// TIA Portal V17 export
// export: Created 2025-03-07T09:17:33.1153197Z, ExportSetting WithDefaults, DisplayName Totally Integrated Automation Portal, DisplayVersion V17 Update 8, DisplayName TIA Portal Openness, DisplayVersion V17 Update 8, DisplayName TIA Portal Version Control Interface, DisplayVersion V17, DisplayName SINAMICS Startdrive Advanced, DisplayVersion V17 SP2, DisplayName SINAMICS Startdrive G110M, G120, G120C, G120D, G120P, G115D, DisplayVersion V17 SP2, DisplayName SINAMICS Startdrive G130, G150, S120, S150, SINAMICS MV, S210, DisplayVersion V17 SP2, DisplayName STEP 7 Professional, DisplayVersion V17 Update 8, DisplayName SINUMERIK ONE STEP 7 Toolbox, DisplayVersion V17 Update 12, DisplayName SINUMERIK 840D sl STEP 7 Toolbox, DisplayVersion V17 Update 12, DisplayName STEP 7 Safety, DisplayVersion V17 Update 6, DisplayName WinCC Advanced, DisplayVersion V17 Update 8
FUNCTION "FC329_CHANNEL_9" : Void   // FC329, LAD
{ S7_Optimized_Access := 'FALSE' }
AUTHOR : ETXETAR
VERSION : 1.0
// stored: AutoNumber false, IsIECCheckEnabled false, SetENOAutomatically false, UDAEnableTagReadback false
   VAR_TEMP
      NC_RESET_CH4 : Bool;
      NC_START_CH4 : Bool;
   END_VAR
BEGIN

REGION Network 1: RESET CHANNEL
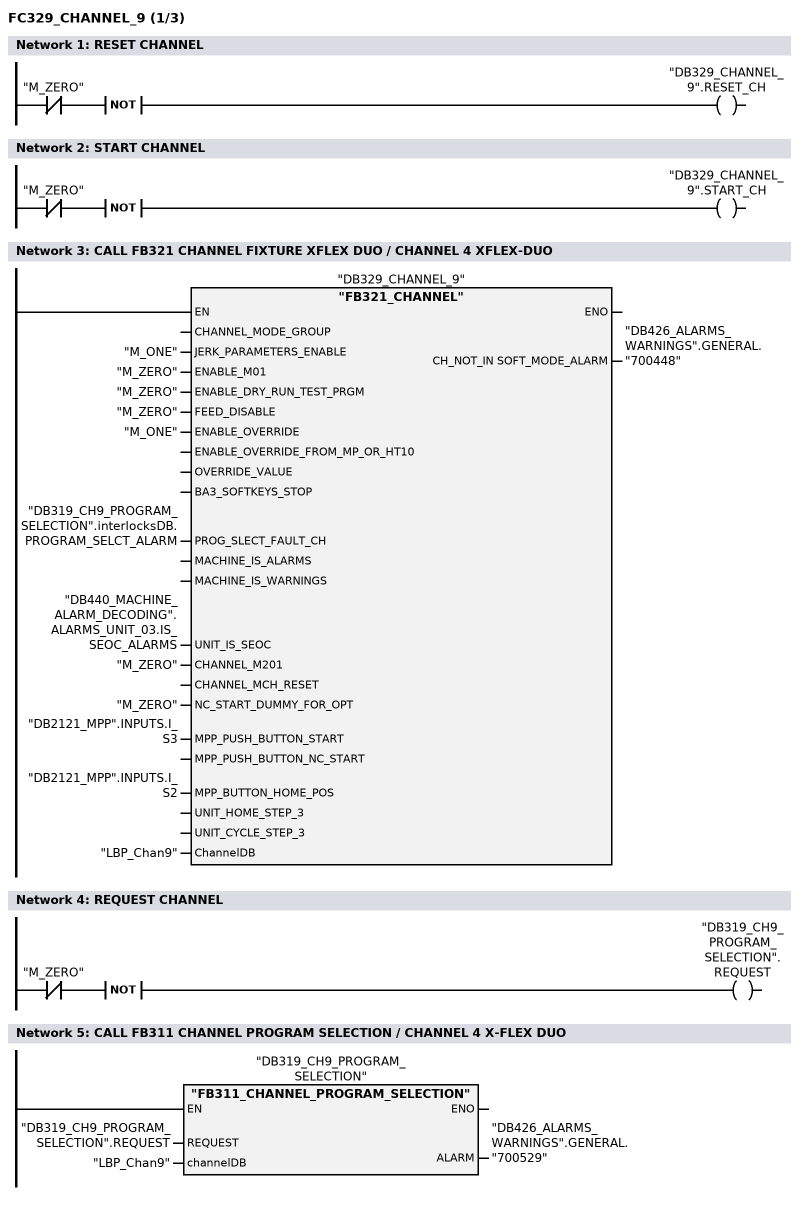
   RUNG wire#powerrail
      I_Contact( "M_ZERO" )
      Not()
      Coil( "DB329_CHANNEL_9".RESET_CH )
   END_RUNG
   // the same network as SCL:
   "DB329_CHANNEL_9".RESET_CH := NOT (NOT "M_ZERO");
END_REGION

REGION Network 2: START CHANNEL
   RUNG wire#powerrail
      I_Contact( "M_ZERO" )
      Not()
      Coil( "DB329_CHANNEL_9".START_CH )
   END_RUNG
   // the same network as SCL:
   "DB329_CHANNEL_9".START_CH := NOT (NOT "M_ZERO");
END_REGION

REGION Network 3: CALL FB321 CHANNEL FIXTURE XFLEX DUO / CHANNEL 4 XFLEX-DUO
   RUNG wire#powerrail
      "DB329_CHANNEL_9"(CHANNEL_MODE_GROUP :=, JERK_PARAMETERS_ENABLE := "M_ONE", ENABLE_M01 := "M_ZERO", ENABLE_DRY_RUN_TEST_PRGM := "M_ZERO", FEED_DISABLE := "M_ZERO", ENABLE_OVERRIDE := "M_ONE", ENABLE_OVERRIDE_FROM_MP_OR_HT10 :=, OVERRIDE_VALUE :=, BA3_SOFTKEYS_STOP :=, PROG_SLECT_FAULT_CH := "DB319_CH9_PROGRAM_SELECTION".interlocksDB.PROGRAM_SELCT_ALARM, MACHINE_IS_ALARMS :=, MACHINE_IS_WARNINGS :=, UNIT_IS_SEOC := "DB440_MACHINE_ALARM_DECODING".ALARMS_UNIT_03.IS_SEOC_ALARMS, CHANNEL_M201 := "M_ZERO", CHANNEL_MCH_RESET :=, NC_START_DUMMY_FOR_OPT := "M_ZERO", MPP_PUSH_BUTTON_START := "DB2121_MPP".INPUTS.I_S3, MPP_PUSH_BUTTON_NC_START :=, MPP_BUTTON_HOME_POS := "DB2121_MPP".INPUTS.I_S2, UNIT_HOME_STEP_3 :=, UNIT_CYCLE_STEP_3 :=, ChannelDB := "LBP_Chan9", "CH_NOT_IN SOFT_MODE_ALARM" => "DB426_ALARMS_WARNINGS".GENERAL."700448")
   END_RUNG
   // the same network as SCL:
   "DB329_CHANNEL_9"(JERK_PARAMETERS_ENABLE := "M_ONE",   // "FB321_CHANNEL"
                     ENABLE_M01 := "M_ZERO",
                     ENABLE_DRY_RUN_TEST_PRGM := "M_ZERO",
                     FEED_DISABLE := "M_ZERO",
                     ENABLE_OVERRIDE := "M_ONE",
                     PROG_SLECT_FAULT_CH := "DB319_CH9_PROGRAM_SELECTION".interlocksDB.PROGRAM_SELCT_ALARM,
                     UNIT_IS_SEOC := "DB440_MACHINE_ALARM_DECODING".ALARMS_UNIT_03.IS_SEOC_ALARMS,
                     CHANNEL_M201 := "M_ZERO",
                     NC_START_DUMMY_FOR_OPT := "M_ZERO",
                     MPP_PUSH_BUTTON_START := "DB2121_MPP".INPUTS.I_S3,
                     MPP_BUTTON_HOME_POS := "DB2121_MPP".INPUTS.I_S2,
                     ChannelDB := "LBP_Chan9",
                     "CH_NOT_IN SOFT_MODE_ALARM" => "DB426_ALARMS_WARNINGS".GENERAL."700448");
END_REGION

REGION Network 4: REQUEST CHANNEL
   RUNG wire#powerrail
      I_Contact( "M_ZERO" )
      Not()
      Coil( "DB319_CH9_PROGRAM_SELECTION".REQUEST )
   END_RUNG
   // the same network as SCL:
   "DB319_CH9_PROGRAM_SELECTION".REQUEST := NOT (NOT "M_ZERO");
END_REGION

REGION Network 5: CALL FB311 CHANNEL PROGRAM SELECTION / CHANNEL 4 X-FLEX DUO
   RUNG wire#powerrail
      "DB319_CH9_PROGRAM_SELECTION"(REQUEST := "DB319_CH9_PROGRAM_SELECTION".REQUEST, channelDB := "LBP_Chan9", ALARM => "DB426_ALARMS_WARNINGS".GENERAL."700529")
   END_RUNG
   // the same network as SCL:
   "DB319_CH9_PROGRAM_SELECTION"(REQUEST := "DB319_CH9_PROGRAM_SELECTION".REQUEST,   // "FB311_CHANNEL_PROGRAM_SELECTION"
                           channelDB := "LBP_Chan9",
                           ALARM => "DB426_ALARMS_WARNINGS".GENERAL."700529");
END_REGION

REGION Network 6: CALL FB301 CHANNEL READ AXES POSITIONS
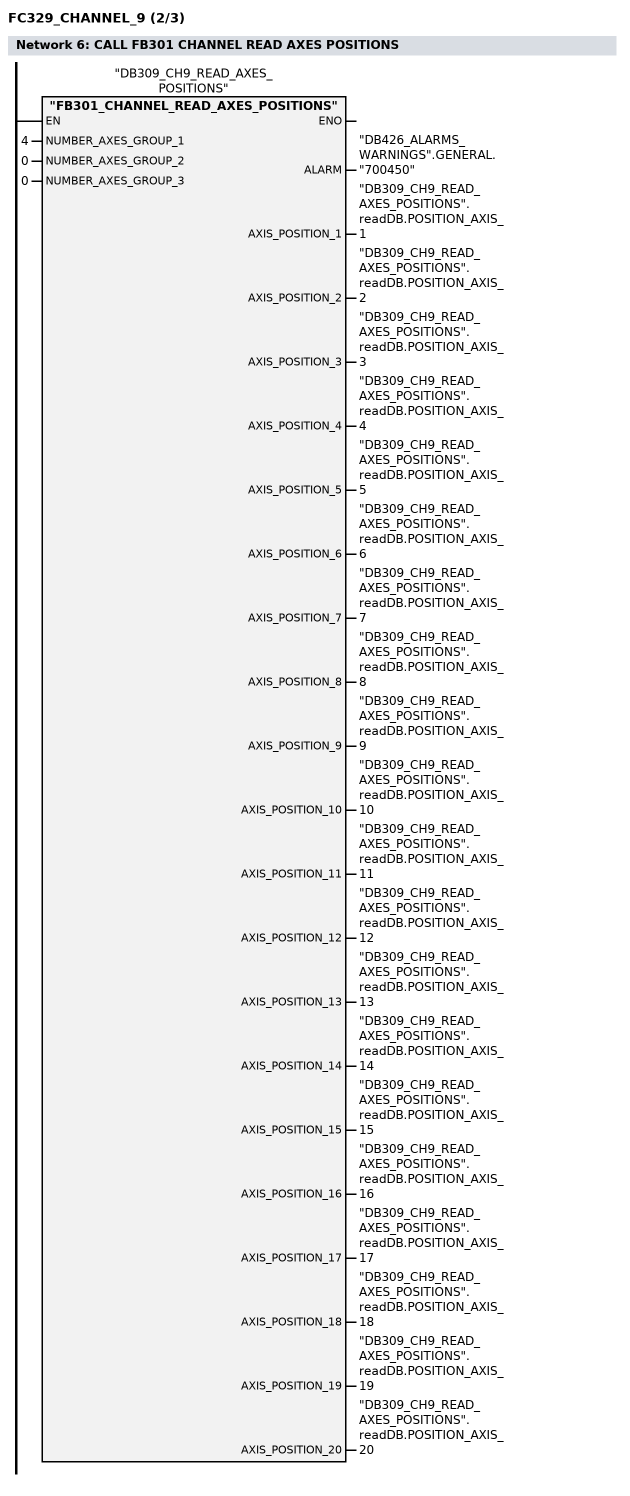
   RUNG wire#powerrail
      "DB309_CH9_READ_AXES_POSITIONS"(NUMBER_AXES_GROUP_1 := 4, NUMBER_AXES_GROUP_2 := 0, NUMBER_AXES_GROUP_3 := 0, ALARM => "DB426_ALARMS_WARNINGS".GENERAL."700450", AXIS_POSITION_1 => "DB309_CH9_READ_AXES_POSITIONS".readDB.POSITION_AXIS_1, AXIS_POSITION_2 => "DB309_CH9_READ_AXES_POSITIONS".readDB.POSITION_AXIS_2, AXIS_POSITION_3 => "DB309_CH9_READ_AXES_POSITIONS".readDB.POSITION_AXIS_3, AXIS_POSITION_4 => "DB309_CH9_READ_AXES_POSITIONS".readDB.POSITION_AXIS_4, AXIS_POSITION_5 => "DB309_CH9_READ_AXES_POSITIONS".readDB.POSITION_AXIS_5, AXIS_POSITION_6 => "DB309_CH9_READ_AXES_POSITIONS".readDB.POSITION_AXIS_6, AXIS_POSITION_7 => "DB309_CH9_READ_AXES_POSITIONS".readDB.POSITION_AXIS_7, AXIS_POSITION_8 => "DB309_CH9_READ_AXES_POSITIONS".readDB.POSITION_AXIS_8, AXIS_POSITION_9 => "DB309_CH9_READ_AXES_POSITIONS".readDB.POSITION_AXIS_9, AXIS_POSITION_10 => "DB309_CH9_READ_AXES_POSITIONS".readDB.POSITION_AXIS_10, AXIS_POSITION_11 => "DB309_CH9_READ_AXES_POSITIONS".readDB.POSITION_AXIS_11, AXIS_POSITION_12 => "DB309_CH9_READ_AXES_POSITIONS".readDB.POSITION_AXIS_12, AXIS_POSITION_13 => "DB309_CH9_READ_AXES_POSITIONS".readDB.POSITION_AXIS_13, AXIS_POSITION_14 => "DB309_CH9_READ_AXES_POSITIONS".readDB.POSITION_AXIS_14, AXIS_POSITION_15 => "DB309_CH9_READ_AXES_POSITIONS".readDB.POSITION_AXIS_15, AXIS_POSITION_16 => "DB309_CH9_READ_AXES_POSITIONS".readDB.POSITION_AXIS_16, AXIS_POSITION_17 => "DB309_CH9_READ_AXES_POSITIONS".readDB.POSITION_AXIS_17, AXIS_POSITION_18 => "DB309_CH9_READ_AXES_POSITIONS".readDB.POSITION_AXIS_18, AXIS_POSITION_19 => "DB309_CH9_READ_AXES_POSITIONS".readDB.POSITION_AXIS_19, AXIS_POSITION_20 => "DB309_CH9_READ_AXES_POSITIONS".readDB.POSITION_AXIS_20)
   END_RUNG
   // the same network as SCL:
   "DB309_CH9_READ_AXES_POSITIONS"(NUMBER_AXES_GROUP_1 := 4,   // "FB301_CHANNEL_READ_AXES_POSITIONS"
                           NUMBER_AXES_GROUP_2 := 0,
                           NUMBER_AXES_GROUP_3 := 0,
                           ALARM => "DB426_ALARMS_WARNINGS".GENERAL."700450",
                           AXIS_POSITION_1 => "DB309_CH9_READ_AXES_POSITIONS".readDB.POSITION_AXIS_1,
                           AXIS_POSITION_2 => "DB309_CH9_READ_AXES_POSITIONS".readDB.POSITION_AXIS_2,
                           AXIS_POSITION_3 => "DB309_CH9_READ_AXES_POSITIONS".readDB.POSITION_AXIS_3,
                           AXIS_POSITION_4 => "DB309_CH9_READ_AXES_POSITIONS".readDB.POSITION_AXIS_4,
                           AXIS_POSITION_5 => "DB309_CH9_READ_AXES_POSITIONS".readDB.POSITION_AXIS_5,
                           AXIS_POSITION_6 => "DB309_CH9_READ_AXES_POSITIONS".readDB.POSITION_AXIS_6,
                           AXIS_POSITION_7 => "DB309_CH9_READ_AXES_POSITIONS".readDB.POSITION_AXIS_7,
                           AXIS_POSITION_8 => "DB309_CH9_READ_AXES_POSITIONS".readDB.POSITION_AXIS_8,
                           AXIS_POSITION_9 => "DB309_CH9_READ_AXES_POSITIONS".readDB.POSITION_AXIS_9,
                           AXIS_POSITION_10 => "DB309_CH9_READ_AXES_POSITIONS".readDB.POSITION_AXIS_10,
                           AXIS_POSITION_11 => "DB309_CH9_READ_AXES_POSITIONS".readDB.POSITION_AXIS_11,
                           AXIS_POSITION_12 => "DB309_CH9_READ_AXES_POSITIONS".readDB.POSITION_AXIS_12,
                           AXIS_POSITION_13 => "DB309_CH9_READ_AXES_POSITIONS".readDB.POSITION_AXIS_13,
                           AXIS_POSITION_14 => "DB309_CH9_READ_AXES_POSITIONS".readDB.POSITION_AXIS_14,
                           AXIS_POSITION_15 => "DB309_CH9_READ_AXES_POSITIONS".readDB.POSITION_AXIS_15,
                           AXIS_POSITION_16 => "DB309_CH9_READ_AXES_POSITIONS".readDB.POSITION_AXIS_16,
                           AXIS_POSITION_17 => "DB309_CH9_READ_AXES_POSITIONS".readDB.POSITION_AXIS_17,
                           AXIS_POSITION_18 => "DB309_CH9_READ_AXES_POSITIONS".readDB.POSITION_AXIS_18,
                           AXIS_POSITION_19 => "DB309_CH9_READ_AXES_POSITIONS".readDB.POSITION_AXIS_19,
                           AXIS_POSITION_20 => "DB309_CH9_READ_AXES_POSITIONS".readDB.POSITION_AXIS_20);
END_REGION

REGION Network 7: CALL FC356 NCK M FIXTURE / CALL FC1182
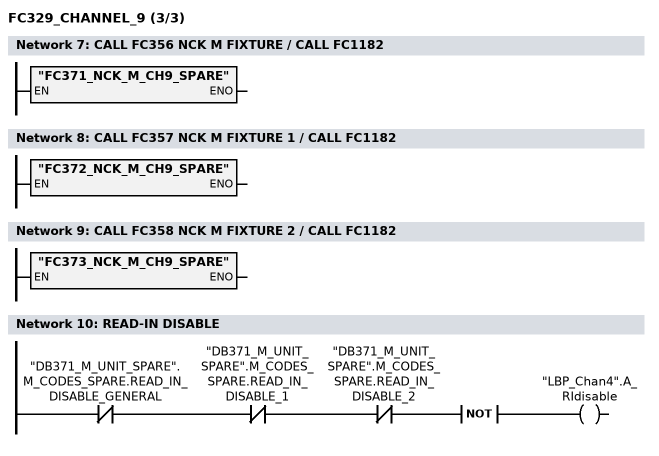
   RUNG wire#powerrail
      "FC371_NCK_M_CH9_SPARE"()
   END_RUNG
   // the same network as SCL:
   "FC371_NCK_M_CH9_SPARE"();
END_REGION

REGION Network 8: CALL FC357 NCK M FIXTURE 1 / CALL FC1182
   RUNG wire#powerrail
      "FC372_NCK_M_CH9_SPARE"()
   END_RUNG
   // the same network as SCL:
   "FC372_NCK_M_CH9_SPARE"();
END_REGION

REGION Network 9: CALL FC358 NCK M FIXTURE 2 / CALL FC1182
   RUNG wire#powerrail
      "FC373_NCK_M_CH9_SPARE"()
   END_RUNG
   // the same network as SCL:
   "FC373_NCK_M_CH9_SPARE"();
END_REGION

REGION Network 10: READ-IN DISABLE
   RUNG wire#powerrail
      I_Contact( "DB371_M_UNIT_SPARE".M_CODES_SPARE.READ_IN_DISABLE_GENERAL )
      I_Contact( "DB371_M_UNIT_SPARE".M_CODES_SPARE.READ_IN_DISABLE_1 )
      I_Contact( "DB371_M_UNIT_SPARE".M_CODES_SPARE.READ_IN_DISABLE_2 )
      Not()
      Coil( "LBP_Chan4".A_RIdisable )
   END_RUNG
   // the same network as SCL:
   "LBP_Chan4".A_RIdisable := NOT (NOT "DB371_M_UNIT_SPARE".M_CODES_SPARE.READ_IN_DISABLE_GENERAL AND NOT "DB371_M_UNIT_SPARE".M_CODES_SPARE.READ_IN_DISABLE_1 AND NOT "DB371_M_UNIT_SPARE".M_CODES_SPARE.READ_IN_DISABLE_2);
END_REGION
END_FUNCTION
